{attribute 'qualified_only'}
{attribute 'strict'}
TYPE E_FestoEmcsStState :
(
	eUnhomed		:=	0,
	eHoming			:=	5,
	eHomingDone		:=	7,
	eUnknown		:=	10,
	eIn				:=	20,
	eOut			:=	30,
	eInter			:=	40,
	eMoveIn			:=	50,
	eSettingIn		:=	55,
	ePlsIn			:=	56,
	eMoveOut		:=	60,
	eSettingOut		:=	65,
	ePlsOut			:=	66,
	eMoveInter		:=	70,
	eSettingInter	:=	75,
	eError			:=	100,
	eResetting		:=	200,
	eEStop			:=	1000						
);
END_TYPE

(* stored: Version 1.1.0.1, ProductVersion 3.1.4026.13, FileIdentifier 3aa5dfecabcda73bce7e53ec0ab3c6ba753e65ea, FileSignature 3acc718aa50c0c86fa1d7aff4111e7ba938a0e587231b23e93a83c68af0a8c777c61f45711ee9912eecc46b1662656c4abcc135deabcbd6438dfa7d410f67259a887c75994c1398365ccdfdd1fb216bd2375c0c8ca91054a5cf454fb6438be242093909b72c44ac6c1784f88d2619de573825dc923337411014c0cb716bc883b967372408a2963d2358b65701d9c937b9af6eb32c11a7c9119dd4ab86d671635f52c8ff66a1cb03ce22403a6e6e97885b64c5a58474a4bcdede007bf0199e6d5a8fca492597d27482ff5c3cdbde1f21839ffbe1d8ed895a7be8cc13acfe4319a479ab5d14dd63513a57df28b0d7596430d3d557de34fd42a40cd524cefb41d19
   DUT E_FestoEmcsStState: Id {8205a6bc-517d-4789-b14f-18b684e43e97} *)
